{attribute 'linkalways'} 
{attribute 'no_explicit_call' := 'This FB is a CLASS and must be accessed using methods or properties'}
{attribute 'enable_dynamic_creation'}
FUNCTION_BLOCK _ETcVnBorderInterpolationMethod EXTENDS EnumDatatypeBase
VAR
	localData : ETcVnBorderInterpolationMethod;
	activeData : REFERENCE TO ETcVnBorderInterpolationMethod;
	enumBaseDatatype : _DINT(localData);
END_VAR

METHOD PRIVATE AddLocalEnumeration
VAR_INPUT
	Enumeration : T_MAXSTRING;
	Value : ETcVnBorderInterpolationMethod;
END_VAR
AddEnumeration(Enumeration, Value);
END_METHOD

PROPERTY PUBLIC Address : PVOID
GET
Address := ADR(activeData);
END_GET
END_PROPERTY

METHOD PUBLIC ClearReference
VAR_INPUT
END_VAR
activeData REF= localData;
SetBaseDatatypeReference();
END_METHOD

METHOD PUBLIC Clone : I_Datatype
VAR
    pClone : POINTER TO _ETcVnBorderInterpolationMethod;
END_VAR
pClone := __NEW(_ETcVnBorderInterpolationMethod(InitialValue := Value));
Clone := pClone^;
END_METHOD

METHOD FB_init : BOOL
VAR_INPUT
	bInitRetains : BOOL; // if TRUE, the retain variables are initialized (warm start / cold start)
	bInCopyCode : BOOL;  // if TRUE, the instance afterwards gets moved into the copy code (online change)
	InitialValue : ETcVnBorderInterpolationMethod;
END_VAR
localData := InitialValue;
AddBaseDatatype(enumBaseDatatype);
ClearReference();

AddLocalEnumeration('TCVN_BIM_CONSTANT', ETcVnBorderInterpolationMethod.TCVN_BIM_CONSTANT);
AddLocalEnumeration('TCVN_BIM_REPLICATE', ETcVnBorderInterpolationMethod.TCVN_BIM_REPLICATE);
AddLocalEnumeration('TCVN_BIM_REFLECT', ETcVnBorderInterpolationMethod.TCVN_BIM_REFLECT);
AddLocalEnumeration('TCVN_BIM_WRAP', ETcVnBorderInterpolationMethod.TCVN_BIM_WRAP);
AddLocalEnumeration('TCVN_BIM_REFLECT_101', ETcVnBorderInterpolationMethod.TCVN_BIM_REFLECT_101);
AddLocalEnumeration('TCVN_BIM_DEFAULT', ETcVnBorderInterpolationMethod.TCVN_BIM_DEFAULT);
AddLocalEnumeration('TCVN_BIM_TRANSPARENT', ETcVnBorderInterpolationMethod.TCVN_BIM_TRANSPARENT);
AddLocalEnumeration('TCVN_BIM_ISOLATED_CONSTANT', ETcVnBorderInterpolationMethod.TCVN_BIM_ISOLATED_CONSTANT);
AddLocalEnumeration('TCVN_BIM_ISOLATED_REPLICATE', ETcVnBorderInterpolationMethod.TCVN_BIM_ISOLATED_REPLICATE);
AddLocalEnumeration('TCVN_BIM_ISOLATED_REFLECT', ETcVnBorderInterpolationMethod.TCVN_BIM_ISOLATED_REFLECT);
AddLocalEnumeration('TCVN_BIM_ISOLATED_WRAP', ETcVnBorderInterpolationMethod.TCVN_BIM_ISOLATED_WRAP);
AddLocalEnumeration('TCVN_BIM_ISOLATED_REFLECT_101', ETcVnBorderInterpolationMethod.TCVN_BIM_ISOLATED_REFLECT_101);
END_METHOD

PROPERTY PUBLIC Identifier : T_MAXSTRING
GET
Identifier := 'ETcVnBorderInterpolationMethod';
END_GET
END_PROPERTY

METHOD IsEnumeratorValueEqual : BOOL
VAR_INPUT
	Enumerator : I_KeyValueForwardEnumerator;
END_VAR
VAR
	storedValue : ETcVnBorderInterpolationMethod;
END_VAR
IF NOT Enumerator.TryGet(storedValue) THEN
	RETURN;
END_IF

IsEnumeratorValueEqual := storedValue = activeData;
END_METHOD

METHOD PUBLIC MakeReferenceTo
VAR_INPUT
	ReferenceTarget : REFERENCE TO ETcVnBorderInterpolationMethod;
END_VAR
activeData REF= ReferenceTarget;
SetBaseDatatypeReference();
END_METHOD

METHOD PROTECTED SetBaseDatatypeReference
VAR_INPUT
END_VAR
enumBaseDatatype.MakeReferenceTo(activeData);
END_METHOD

PROPERTY PUBLIC Size : UDINT
GET
Size := SIZEOF(activeData);
END_GET
END_PROPERTY

METHOD TryMakeReferenceTo : BOOL
VAR_INPUT
	Target : I_Datatype;
END_VAR
VAR
	pTargetData : POINTER TO ETcVnBorderInterpolationMethod;
END_VAR
IF NOT IsEquivalentTo(Target) THEN
	RETURN;
END_IF

pTargetData := Target.Address;
activeData REF= pTargetData^;
SetBaseDatatypeReference();
TryMakeReferenceTo := TRUE;
END_METHOD

PROPERTY PUBLIC Value : ETcVnBorderInterpolationMethod
GET
Value := activeData;
END_GET
SET
activeData := Value;
END_SET
END_PROPERTY

END_FUNCTION_BLOCK

(* stored: Version 1.1.0.1, ProductVersion 3.1.4024.13
   POU _ETcVnBorderInterpolationMethod: Id {0cb2776b-3fd6-4868-8627-c717ad33cae1}, SpecialFunc None
   Folder Core: Id {4c585a1a-77fb-098f-29c3-b1271f37f3b7}
   Folder Protected: Id {e2b73acf-685b-0cb0-3eab-47636794efd8}
   Folder Customize: Id {f0f55a4a-ea82-057d-2031-164e427b7bbf}
   Folder Constructor: Id {fc51c54b-d9f3-4f87-acf0-02f60cc271a1}
   Folder Private: Id {5a14e1f2-0b2a-4ea3-b139-2ce03e7b4a8b}
   Folder Protected: Id {c53f1e99-7a09-40de-a834-425a12b672c0}
   Method AddLocalEnumeration: Id {7f73779e-6ef6-45bc-83f0-c146700fce05}
   Property Address: Id {4da06f9d-4d41-069e-06be-18f0dcda3abb}
   Get Get: Id {2a83a418-d9bd-00eb-15ee-6b68aa635311}
   Method ClearReference: Id {f6490e81-67d5-01ab-0d33-1704813bc111}
   Method Clone: Id {16646000-fb57-4a7e-b571-d03ffad8bbdd}
   Method FB_init: Id {7d82cf3b-d344-48c5-b15f-768fee5a5a3e}
   Property Identifier: Id {dd6cd104-b4d1-407d-94ca-c4c8d266aae2}
   Get Get: Id {23df3589-1fa5-4eae-bcfe-04b3f9796e2a}
   Method IsEnumeratorValueEqual: Id {9d06e305-bb16-49c3-8d9e-6f24c5fae3f7}
   Method MakeReferenceTo: Id {859a5dfb-39b4-4b61-8a3f-fec71cc79ceb}
   Method SetBaseDatatypeReference: Id {c2e8b82b-3041-0391-3bb3-1e06f93e23f2}
   Property Size: Id {b70e1a8d-4b64-011c-30ec-5536c5c0bb3c}
   Get Get: Id {66e22b21-1f70-0841-00c5-c5d0ce40f25e}
   Method TryMakeReferenceTo: Id {9b9ce214-95a2-47b2-b8aa-a37c0a0ea0b9}
   Property Value: Id {b9bd6223-e1da-4e6f-8751-50c1bef71c79}
   Get Get: Id {d5fa5e93-b39b-4e27-aac1-293c68aff6e7}
   Set Set: Id {cc15d6da-de1e-41dc-9271-322d307d2790} *)
